(* Schneider Machine Expert - Basic project Tank_Level_AI_v11, file version 3.0.0.0 *)
(* ProjectInformations: Name=Tank_Level_AI_v11 *)

HARDWARE
  Cpu 0: TM221CE24T
  EthernetConfiguration: NetworkName=M221, IpAllocationMode=ByDhcp, IpAddress=192.168.1.10, SubnetMask=255.255.255.0
  SerialLineConfiguration: Baud=Baud19200, Parity=ParityEven, DataBits=DataBits8, StopBits=StopBits1, PhysicalMedium=PhysicalMediumRs485, TransmissionMode=TransmissionModeModbusRtu, SlaveId=1, Addressing=SlaveAddressing
  MastTask: UsePeriodScanMode=false, PeriodScan=100
  FastTask: Period=255
  CpuBehavior: StartingMode=StartAsPreviousState, AutoSaveRamOnEeprom=true, WatchdogPeriod=250

SYMBOLS  (address, symbol, comment, settings)
  %M0       PUMP_RUN  "Pump running flag"
  %M1       LEVEL_LOW  "Tank level low flag"
  %M2       LEVEL_HIGH  "Tank level high flag"
  %I0.2     ESTOP
  %Q0.0     INLET_VALVE
  %Q0.1     OUTLET_VALVE

POU Main Program
  (* SectionNumber=1 *)

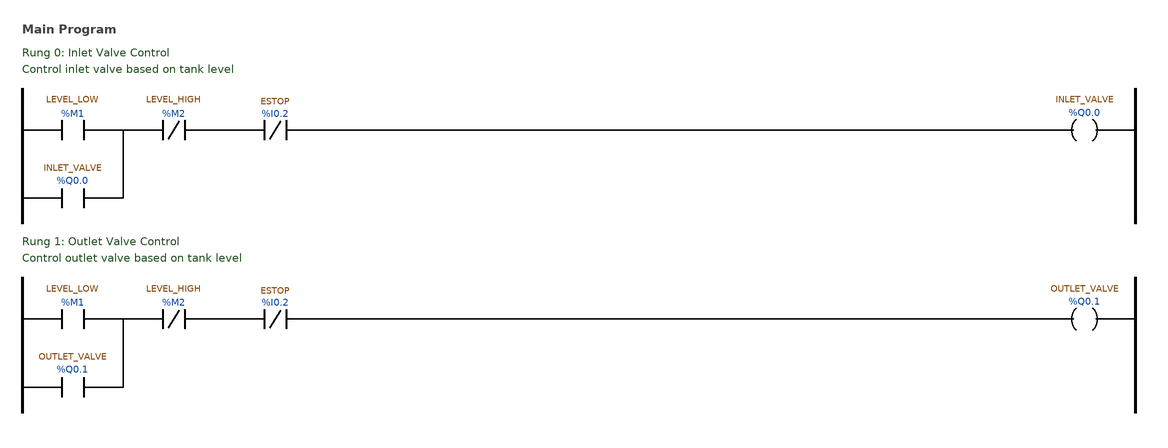

// Rung 0: Inlet Valve Control
// Control inlet valve based on tank level
  LD %M1                  (* LEVEL_LOW *)
  OR %Q0.0                (* INLET_VALVE *)
  ANDN %M2                (* LEVEL_HIGH *)
  ANDN %I0.2              (* ESTOP *)
  ST %Q0.0                (* INLET_VALVE *)
  // as ST:
  //   INLET_VALVE := (LEVEL_LOW OR INLET_VALVE) AND NOT LEVEL_HIGH AND NOT ESTOP;

// Rung 1: Outlet Valve Control
// Control outlet valve based on tank level
  LD %M1                  (* LEVEL_LOW *)
  OR %Q0.1                (* OUTLET_VALVE *)
  ANDN %M2                (* LEVEL_HIGH *)
  ANDN %I0.2              (* ESTOP *)
  ST %Q0.1                (* OUTLET_VALVE *)
  // as ST:
  //   OUTLET_VALVE := (LEVEL_LOW OR OUTLET_VALVE) AND NOT LEVEL_HIGH AND NOT ESTOP;

// Rung 2: High Level Detection
// Set high level flag when tank is full
  LD [%IW1.0>=10000]
  ST %M2                  (* LEVEL_HIGH *)
  // as ST:
  //   LEVEL_HIGH := %IW1.0>=10000;
  (* the ladder stored for this rung does not match its IL; not drawn *)

// Rung 3: Low Level Detection
// Set low level flag when tank is empty
  LD [%IW1.0<=3000]
  ST %M1                  (* LEVEL_LOW *)
  // as ST:
  //   LEVEL_LOW := %IW1.0<=3000;
  (* the ladder stored for this rung does not match its IL; not drawn *)
